FUNCTION_BLOCK IED87 (* Extracted Composite Function Block Type *)
  (* Version 3/31/2017, bdowdesw *)
  PACKAGE Main;
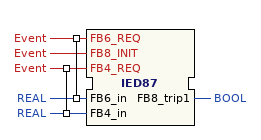
  EVENT_INPUT
    FB6_REQ WITH FB6_in; (* Normal Execution Request *)
    FB8_INIT; (* Initialization Request *)
    FB4_REQ WITH FB4_in; (* Normal Execution Request *)
  END_EVENT
  VAR_INPUT
    FB6_in : REAL; (* Input event qualifier *)
    FB4_in : REAL; (* Input event qualifier *)
  END_VAR
  VAR_OUTPUT
    FB8_trip1 : BOOL;
  END_VAR
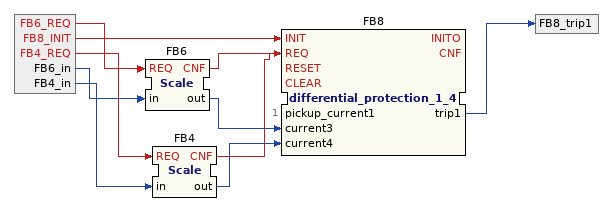
  FBS
    FB6 : Scale;
    FB4 : Scale;
    FB8 : differential_protection_1_4(pickup_current1 := 1);
  END_FBS
  EVENT_CONNECTIONS
    FB6.CNF TO FB8.REQ;
    FB4.CNF TO FB8.REQ;
    FB6_REQ TO FB6.REQ;
    FB8_INIT TO FB8.INIT;
    FB4_REQ TO FB4.REQ;
  END_CONNECTIONS
  DATA_CONNECTIONS
    FB6.out TO FB8.current3;
    FB4.out TO FB8.current4;
    FB6_in TO FB6.in;
    FB8.trip1 TO FB8_trip1;
    FB4_in TO FB4.in;
  END_CONNECTIONS
END_FUNCTION_BLOCK
